PROGRAM MAIN
VAR
	a:INT;
	b:INT;
	c:INT;
END_VAR

END_PROGRAM

(* stored: Version 1.1.0.1, ProductVersion 3.1.4024.3
   POU MAIN: Id {055e7c0c-b0d7-4752-aa06-12966b43f93a}, SpecialFunc None *)
